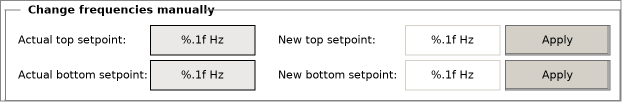
VISUALIZATION VISU_HydraulicsChangeFrequencies  // 622x102
VAR_IN_OUT
	ref : Hydraulics;
    widget : HydraulicsWidget;
END_VAR
    Label (25,0 175x20), "Change frequencies manually"
    Polyline (20,10) (5,10) (5,100) (620,100) (620,10) (205,10)
    Button (505,25 105x30), "Apply", input disabled if: ref.parts.top.processes.changeFrequencySetpoint.statuses.enabledStatus.disabled
        OnMouseClick: execute { ref.parts.top.processes.changeFrequencySetpoint.do_request := TRUE; }
    Label (15,25 110x30), "Actual top setpoint:"
    Label (15,60 130x30), "Actual bottom setpoint:"
    Rectangle (150,25 105x30), "%.1f Hz", text variable: ref.parts.top.driveSetpoint.hertz.value
    Rectangle (150,60 105x30), "%.1f Hz", text variable: ref.parts.bottom.driveSetpoint.hertz.value
    Textfield (405,25 95x30), "%.1f Hz", text variable: ref.parts.top.processes.changeFrequencySetpoint.set.setpoint, input disabled if: ref.parts.top.processes.changeFrequencySetpoint.statuses.enabledStatus.disabled
        OnMouseClick: write the text variable via VisuDialogs.Numpad
    Label (275,25 120x30), "New top setpoint:"
    Label (275,60 130x30), "New bottom setpoint:"
    Button (505,60 105x30), "Apply", input disabled if: ref.parts.bottom.processes.changeFrequencySetpoint.statuses.enabledStatus.disabled
        OnMouseClick: execute { ref.parts.bottom.processes.changeFrequencySetpoint.do_request := TRUE; }
    Textfield (405,60 95x30), "%.1f Hz", text variable: ref.parts.bottom.processes.changeFrequencySetpoint.set.setpoint, input disabled if: ref.parts.bottom.processes.changeFrequencySetpoint.statuses.enabledStatus.disabled
        OnMouseClick: write the text variable via VisuDialogs.Numpad
END_VISUALIZATION

(* stored: Version 1.1.0.1, ProductVersion 3.1.4018.5
   Visu VISU_HydraulicsChangeFrequencies: Id {339ad3e0-45d7-4245-96be-f2eefb69fe31} *)
